(* CoDeSys 2.3 export: GLOBAL_VARIABLES.EXP *)

(* Global variable list: Global_Variables *)
VAR_GLOBAL
    hoz: INT;
    ver: INT;
	MAPA: ARRAY[0..20, 0..15] OF BOOL;
	Mapa_Punkty: ARRAY[0..20, 0..15] OF BOOL;
	Wolne_Prawo: BOOL;
	Wolne_Lewo: BOOL;
	Wolne_Dol: BOOL;
	Wolne_Gora: BOOL;
	Otwarte: BOOL := TRUE;
	Kierunek: INT := 1;
 B_Prawo : BOOL := TRUE;
   B_Lewo  : BOOL;
   B_Dol   : BOOL;
   B_Gora  : BOOL;

END_VAR
